Fanuc TP program (LS listing): message6.ls

/PROG  MESSAGE6	  Macro
/ATTR
OWNER		= MNEDITOR;
COMMENT		= "USER MESSAGE";
PROG_SIZE	= 351;
CREATE		= DATE 21-07-12  TIME 16:24:48;
MODIFIED	= DATE 22-05-17  TIME 09:36:08;
FILE_NAME	= MESSAGE5;
VERSION		= 0;
LINE_COUNT	= 2;
MEMORY_SIZE	= 731;
PROTECT		= READ_WRITE;
TCD:  STACK_SIZE	= 0,
      TASK_PRIORITY	= 50,
      TIME_SLICE	= 0,
      BUSY_LAMP_OFF	= 0,
      ABORT_REQUEST	= 0,
      PAUSE_REQUEST	= 7;
DEFAULT_GROUP	= *,*,*,*,*;
CONTROL_CODE	= 00000000 00000000;
/APPL
/APPL

AUTO_SINGULARITY_HEADER;
  ENABLE_SINGULARITY_AVOIDANCE   : FALSE;
/MN
   1:  CALL MESSAGE20    ;
   2:  CALL FAULT_MESSAGE('Robot is in step mode.','Press the step button','on the robot teach pendant','to run continuous mode.') ;
/POS
/END
